Yaskawa INFORM job: R2_W57-58-A2(80,180)AW-OK.JBI

/JOB
//NAME R2_W57-58-A2(80,180)AW-OK
///FOLDERNAME AWOK
//POS
///NPOS 64,64,0,3,0,0
///TOOL 0
///POSTYPE PULSE
///PULSE
C00000=142653,16598,-52845,-13185,75828,-55165
C00001=107308,79936,29099,21901,57164,-61647
C00002=107309,74973,39858,24593,48699,-63677
C00003=107310,74708,42040,25145,47351,-64051
C00004=107310,74641,42958,25380,46806,-64207
C00005=107310,74578,44264,25719,46049,-64430
C00006=108285,73900,43455,24894,45893,-63988
C00007=107310,74578,44264,25719,46049,-64430
C00008=107310,74641,42958,25380,46806,-64207
C00009=107309,74627,42816,25348,46880,-64186
C00010=107309,74562,43948,25641,46217,-64380
C00011=107309,74627,42816,25348,46880,-64186
C00012=107310,74641,42958,25380,46806,-64207
C00013=107309,78322,31127,14468,73984,-64784
C00014=103975,94985,53278,24753,70738,-64932
C00015=104439,94509,52669,24536,70723,-64762
C00016=103279,95651,52516,24942,71677,-64986
C00017=107309,78322,31127,14468,73984,-64784
C00018=107310,80743,28406,14295,76815,-64446
C00019=107308,89822,23730,14034,84139,-63602
C00020=120730,109686,61376,15286,111101,-79643
C00021=120730,108445,63352,15082,109309,-79882
C00022=120730,108030,64247,15004,108570,-79978
C00023=120730,108143,63990,15025,108780,-79951
C00024=120730,107748,64935,14946,108020,-80049
C00025=120730,108143,63990,15025,108780,-79951
C00026=120730,108030,64247,15004,108570,-79978
C00027=120730,105951,60555,15128,109734,-79825
C00028=120730,103678,57575,15202,110377,-79740
C00029=120730,108267,63605,15056,109070,-79913
C00030=120730,108030,64247,15004,108570,-79978
C00031=120732,107362,65241,24315,60633,-68503
C00032=120732,107337,65208,24312,60639,-68501
C00033=121379,107353,65229,23949,60452,-68282
C00034=120732,107337,65208,24312,60639,-68501
C00035=120731,107368,65249,24315,60631,-68503
C00036=120731,107425,65323,24319,60616,-68507
C00037=120731,107410,65303,24318,60620,-68506
C00038=120731,107389,65277,24316,60625,-68505
C00039=145565,127861,77876,-5846,97918,-52225
C00040=146001,127366,81238,-5857,95636,-51975
C00041=145948,126998,81756,-5845,95125,-51971
C00042=146361,130124,85639,-5881,94377,-51796
C00043=146204,126945,81045,-5878,95553,-51903
C00044=132042,124336,80430,-4231,93732,-56517
C00045=132042,125260,78662,-4244,95290,-56570
C00046=153059,90356,29758,-7012,108738,-50365
C00047=152481,84969,31810,-6779,104690,-50317
C00048=147780,134592,93634,-6010,91868,-51204
C00049=147631,130708,88050,-6006,93291,-51322
C00050=162988,74642,21528,-7917,106571,-47014
C00051=163599,74245,21048,-7983,106717,-46823
C00052=162188,77497,22810,-7871,107174,-47313
C00053=147595,132318,87700,-6013,94325,-51384
C00054=134156,132683,88199,-4480,93353,-55799
C00055=132043,128288,75738,-4285,98637,-56683
C00056=132043,124281,80353,-4232,93750,-56517
C00057=134386,134735,95665,-4490,89836,-55597
C00058=134168,130923,90179,-4469,91237,-55720
C00059=140932,95843,44959,-5395,101401,-53902
C00060=143847,69618,12121,-11281,94579,-53544
C00061=147608,43855,-23769,-15212,95284,-53260
C00062=142653,16598,-52845,-13185,75828,-55165
C00063=93296,-8034,-64184,-13230,75773,-55134
BC00000=299827,326488,1072504
BC00001=280350,208884,1075175
BC00002=279887,208793,1075175
BC00003=276067,203889,1075175
BC00004=274540,201927,1075175
BC00005=274520,201476,1075175
BC00006=274520,201476,1075175
BC00007=274520,201476,1075175
BC00008=274540,201927,1075175
BC00009=280431,200366,1075175
BC00010=280431,200366,1075175
BC00011=280431,200366,1075175
BC00012=274540,201927,1075175
BC00013=277320,168503,1075175
BC00014=274026,164767,1075175
BC00015=274026,164767,1075175
BC00016=274026,164767,1075175
BC00017=277320,168503,1075175
BC00018=269646,175108,1075175
BC00019=274616,178947,1075175
BC00020=250084,179282,1075175
BC00021=248393,182772,1075175
BC00022=247717,184168,1075175
BC00023=247705,179923,1075175
BC00024=247705,179923,1075175
BC00025=247705,179923,1075175
BC00026=247717,184168,1075175
BC00027=255215,184460,1075175
BC00028=255215,184460,1075175
BC00029=255215,184460,1075175
BC00030=247717,184168,1075175
BC00031=275847,263556,995153
BC00032=275767,262446,963418
BC00033=275767,262446,963418
BC00034=275767,262446,963418
BC00035=275887,264563,1002604
BC00036=266423,262144,1017568
BC00037=268126,262311,1008695
BC00038=272492,264160,1009079
BC00039=398174,127384,1075175
BC00040=398174,128102,1075175
BC00041=398174,128390,1075175
BC00042=398174,128390,1075175
BC00043=398174,128390,1075175
BC00044=307557,170717,1071451
BC00045=307557,170717,1071451
BC00046=344898,147714,1075175
BC00047=344898,147714,1075175
BC00048=380696,148720,1075175
BC00049=380696,148720,1075175
BC00050=344898,147714,1075175
BC00051=344898,147714,1075175
BC00052=344898,147714,1075175
BC00053=359794,167940,1075175
BC00054=307064,181639,1075175
BC00055=307557,170717,1071451
BC00056=307557,170717,1071451
BC00057=304467,182645,1075175
BC00058=304467,182645,1075175
BC00059=307557,170717,1071451
BC00060=307557,170717,1071451
BC00061=307557,170717,1071451
BC00062=299827,326488,1072504
BC00063=215214,386961,1072501
///POSTYPE BASE
///RECTAN
///RCONF 0,0,0,0,0,0,0,0,0,0,0,0,0,0,0,0,0,0,0,0,0,0,0,0
P00006=0.222,-3.123,-1.508,0.0000,0.0000,0.0000
P00020=2.715,4.999,8.452,0.0000,0.0000,0.0000
P00021=-0.225,-6.128,-0.405,0.0000,0.0000,0.0000
//INST
///DATE 2023/11/16 10:54
///ATTR SC,RW
///GROUP1 RB1,BS1
NOP
'r2_W57-58-A2(80,180)
'Path S1102
SFTOF
MOVJ C00000 BC00000 VJ=20.00
MOVJ C00001 BC00001 VJ=20.00
MOVJ C00002 BC00002 VJ=20.00
MOVL C00003 BC00003 V=100.0
MOVL C00004 BC00004 V=100.0
MOVL C00005 BC00005 V=60.0
REFP 3 C00006 BC00006
CALL JOB:SEARCH-R1
SET P020 P006
SFTON P020
MOVL C00007 BC00007 V=60.0
MOVL C00008 BC00008 V=100.0
MOVL C00009 BC00009 V=60.0
REFP 3 C00010 BC00010
CALL JOB:SEARCH-R1
SET P020 P006
SFTON P020
MOVL C00011 BC00011 V=60.0
MOVL C00012 BC00012 V=100.0
MOVL C00013 BC00013 V=100.0
MOVL C00014 BC00014 V=60.0
REFP 3 C00015 BC00015
CALL JOB:SEARCH-R1
SET P020 P006
SFTON P020
MOVL C00016 BC00016 V=60.0
MOVL C00017 BC00017 V=100.0
MOVL C00018 BC00018 V=100.0
MOVL C00019 BC00019 V=100.0
'Path S1103
SFTOF
MOVJ C00020 BC00020 VJ=20.00 ENWAIT DIS=250.0
DOUT OG#(200) 12
MOVL C00021 BC00021 V=100.0
MOVL C00022 BC00022 V=100.0
MOVL C00023 BC00023 V=60.0
REFP 3 C00024 BC00024
CALL JOB:SEARCH-R1
SET P021 P006
SFTON P021
MOVL C00025 BC00025 V=60.0
MOVL C00026 BC00026 V=100.0
MOVL C00027 BC00027 V=60.0
REFP 3 C00028 BC00028
CALL JOB:SEARCH-R1
SET P021 P006
SFTON P021
MOVL C00029 BC00029 V=60.0
MOVL C00030 BC00030 V=100.0
MOVL C00031 BC00031 V=100.0
MOVL C00032 BC00032 V=60.0
REFP 3 C00033 BC00033
CALL JOB:SEARCH-R1
SET P021 P006
SFTON P021
MOVL C00034 BC00034 V=60.0
MOVL C00035 BC00035 V=100.0
MOVL C00036 BC00036 V=100.0
MOVL C00037 BC00037 V=100.0
MOVL C00038 BC00038 V=100.0
'Path W1104
SFTOF
SFTON P020
MOVJ C00039 BC00039 VJ=20.00
MOVL C00040 BC00040 V=100.0
MOVL C00041 BC00041 V=100.0 PL=0
REFP 1 C00042 BC00042
REFP 2 C00043 BC00043
MACRO1 MJ#(0) ARGF10
ARCON
MOVL C00044 BC00044 V=14.2
ARCOF
MOVL C00045 BC00045 V=100.0
SFTOF
'Path W1105
SFTOF
SFTON P020
MOVJ C00046 BC00046 VJ=20.00
DOUT OG#(200) 13
MOVL C00047 BC00047 V=100.0 PL=0
REFP 1 C00048 BC00048
REFP 2 C00049 BC00049
MACRO1 MJ#(0) ARGF10
ARCON
MOVL C00050 BC00050 V=15.0
MOVL C00051 BC00051 V=15.0
ARCOF
MOVL C00052 BC00052 V=100.0
MOVL C00053 BC00053 V=100.0
SFTOF
'Path W1106
SFTOF
SFTON P021
MOVJ C00054 BC00054 VJ=20.00
MOVL C00055 BC00055 V=100.0
MOVL C00056 BC00056 V=100.0 PL=0
REFP 1 C00057 BC00057
REFP 2 C00058 BC00058
MACRO1 MJ#(0) ARGF10
ARCON
MOVL C00059 BC00059 V=15.0
ARCOF
MOVL C00060 BC00060 V=100.0
MOVL C00061 BC00061 V=100.0
DOUT OG#(200) 14
SFTOF
'Path W1107
SFTOF
SFTON P021
SFTOF
MOVJ C00062 BC00062 VJ=20.00
MOVJ C00063 BC00063 VJ=20.00
END
